# B&R Automation Studio project RobotNewEra (part 4)

```c
	// prepare
	int bol = m_brightleft ? m_elxlist.GetSize() : -1;
	int stp = m_brightleft ? -1 : 1;
	int eol = m_brightleft ? -1 : m_elxlist.GetSize();

	// from last
	int n = eol - stp;

	while(n != bol && ! m_elxlist[n]->MatchNext(pContext))
		n -= stp;

	if(n != bol)
		n += stp;
	else
		return 0;

	// match rest
	while(n != eol)
	{
		if(m_elxlist[n]->Match(pContext))
		{
			n += stp;
		}
		else
		{
			n -= stp;

			while(n != bol && ! m_elxlist[n]->MatchNext(pContext))
				n -= stp;

			if(n != bol)
				n += stp;
			else
				return 0;
		}
	}

	return 1;
}

// mresult.cpp: implementation of the MatchResult class.
//
template <int x> MatchResultT <x> :: MatchResultT(CContext * pContext, int nMaxNumber)
{
	if(pContext != 0)
	{
		m_result.Prepare(nMaxNumber * 2 + 3, -1);

		// matched
		m_result[0] = 1;
		m_result[1] = nMaxNumber;

		for(int n = 0; n <= nMaxNumber; n++)
		{
			int index = pContext->m_captureindex[n];
			//if( index < 0 ) continue;
			if( ! CBracketElxT<char>::CheckCaptureIndex(index, pContext, n) ) continue;

			// check enclosed
			int pos1 = pContext->m_capturestack[index + 1];
			int pos2 = pContext->m_capturestack[index + 2];

			// info
			m_result[n*2 + 2] = pos1 < pos2 ? pos1 : pos2;
			m_result[n*2 + 3] = pos1 < pos2 ? pos2 : pos1;
		}
	}
}

template <int x> inline int MatchResultT <x> :: IsMatched() const
{
	return m_result.At(0, 0);
}

template <int x> inline int MatchResultT <x> :: MaxGroupNumber() const
{
	return m_result.At(1, 0);
}

template <int x> inline int MatchResultT <x> :: GetStart() const
{
	return m_result.At(2, -1);
}

template <int x> inline int MatchResultT <x> :: GetEnd() const
{
	return m_result.At(3, -1);
}

template <int x> inline int MatchResultT <x> :: GetGroupStart(int nGroupNumber) const
{
	return m_result.At(2 + nGroupNumber * 2, -1);
}

template <int x> inline int MatchResultT <x> :: GetGroupEnd(int nGroupNumber) const
{
	return m_result.At(2 + nGroupNumber * 2 + 1, -1);
}

template <int x> MatchResultT <x> & MatchResultT <x> :: operator = (const MatchResultT <x> & result)
{
	m_result.Restore(0);
	if(result.m_result.GetSize() > 0) m_result.Append(result.m_result.GetBuffer(), result.m_result.GetSize());

	return *this;
}

// posselx.cpp: implementation of the CPossessiveElx class.
//
template <int x> CPossessiveElxT <x> :: CPossessiveElxT(ElxInterface * pelx, int nmin, int nmax) : CGreedyElxT <x> (pelx, nmin, nmax)
{
}

template <int x> int CPossessiveElxT <x> :: Match(CContext * pContext) const
{
	int nbegin = pContext->m_nCurrentPos;
	int nsize  = pContext->m_stack.GetSize();
	int ncsize = pContext->m_capturestack.GetSize();
	int bsucc  = 1;

	// match
	if( ! CRepeatElxT <x> :: MatchFixed(pContext) )
	{
		bsucc = 0;
	}
	else
	{
		while( ! CGreedyElxT <x> :: MatchVart(pContext) )
		{
			if( ! CRepeatElxT <x> :: MatchNextFixed(pContext) )
			{
				bsucc = 0;
				break;
			}
		}
	}

	// status
	pContext->m_stack.Restore(nsize);

	if( bsucc )
	{
		pContext->m_stack.Push(nbegin);
		pContext->m_stack.Push(ncsize);
	}

	return bsucc;
}

template <int x> int CPossessiveElxT <x> :: MatchNext(CContext * pContext) const
{
	int nbegin = 0, ncsize = 0;

	pContext->m_stack.Pop(ncsize);
	pContext->m_stack.Pop(nbegin);

	pContext->m_capturestack.Restore(ncsize);
	pContext->m_nCurrentPos = nbegin;

	return 0;
}

// reluctx.cpp: implementation of the CReluctantElx class.
//
template <int x> CReluctantElxT <x> :: CReluctantElxT(ElxInterface * pelx, int nmin, int nmax) : CRepeatElxT <x> (pelx, nmin)
{
	m_nvart = nmax - nmin;
}

template <int x> int CReluctantElxT <x> :: Match(CContext * pContext) const
{
	if( ! CRepeatElxT <x> :: MatchFixed(pContext) )
		return 0;

	while( ! MatchVart(pContext) )
	{
		if( ! CRepeatElxT <x> :: MatchNextFixed(pContext) )
			return 0;
	}

	return 1;
}

template <int x> int CReluctantElxT <x> :: MatchNext(CContext * pContext) const
{
	if( MatchNextVart(pContext) )
		return 1;

	if( ! CRepeatElxT <x> :: MatchNextFixed(pContext) )
		return 0;

	while( ! MatchVart(pContext) )
	{
		if( ! CRepeatElxT <x> :: MatchNextFixed(pContext) )
			return 0;
	}

	return 1;
}

template <int x> int CReluctantElxT <x> :: MatchVart(CContext * pContext) const
{
	pContext->m_stack.Push(0);

	return 1;
}

template <int x> int CReluctantElxT <x> :: MatchNextVart(CContext * pContext) const
{
	int n = 0, nbegin = pContext->m_nCurrentPos;

	pContext->m_stack.Pop(n);

	if(n < m_nvart && CRepeatElxT <x> :: m_pelx->Match(pContext))
	{
		while(pContext->m_nCurrentPos == nbegin)
		{
			if( ! CRepeatElxT <x> :: m_pelx->MatchNext(pContext) ) break;
		}

		if(pContext->m_nCurrentPos != nbegin)
		{
			n ++;

			pContext->m_stack.Push(nbegin);
			pContext->m_stack.Push(n);

			return 1;
		}
	}

	while(n > 0)
	{
		pContext->m_stack.Pop(nbegin);

		while( CRepeatElxT <x> :: m_pelx->MatchNext(pContext) )
		{
			if(pContext->m_nCurrentPos != nbegin)
			{
				pContext->m_stack.Push(nbegin);
				pContext->m_stack.Push(n);

				return 1;
			}
		}

		n --;
	}

	return 0;
}

// repeatx.cpp: implementation of the CRepeatElx class.
//
template <int x> CRepeatElxT <x> :: CRepeatElxT(ElxInterface * pelx, int ntimes)
{
	m_pelx   = pelx;
	m_nfixed = ntimes;
}

template <int x> int CRepeatElxT <x> :: Match(CContext * pContext) const
{
	return MatchFixed(pContext);
}

template <int x> int CRepeatElxT <x> :: MatchNext(CContext * pContext) const
{
	return MatchNextFixed(pContext);
}

template <int x> int CRepeatElxT <x> :: MatchFixed(CContext * pContext) const
{
	if(m_nfixed == 0)
		return 1;

	int n = 0;

	while(n < m_nfixed)
	{
		if(m_pelx->Match(pContext))
		{
			n ++;
		}
		else
		{
			n --;

			while(n >= 0 && ! m_pelx->MatchNext(pContext))
				n --;

			if(n >= 0)
				n ++;
			else
				return 0;
		}
	}

	return 1;
}

template <int x> int CRepeatElxT <x> :: MatchNextFixed(CContext * pContext) const
{
	if(m_nfixed == 0)
		return 0;

	// from last
	int n = m_nfixed - 1;

	while(n >= 0 && ! m_pelx->MatchNext(pContext))
		n --;

	if(n >= 0)
		n ++;
	else
		return 0;

	// match rest
	while(n < m_nfixed)
	{
		if(m_pelx->Match(pContext))
		{
			n ++;
		}
		else
		{
			n --;

			while(n >= 0 && ! m_pelx->MatchNext(pContext))
				n --;

			if(n >= 0)
				n ++;
			else
				return 0;
		}
	}

	return 1;
}

// Regexp
typedef CRegexpT <char> CRegexpA;
typedef CRegexpT <unsigned short> CRegexpW;

#if defined(_UNICODE) || defined(UNICODE)
	typedef CRegexpW CRegexp;
#else
	typedef CRegexpA CRegexp;
#endif

#endif//__DEELX_REGEXP__H__
```

### Package Logical/MotionHandling - Motion Handling

### MotionGlobal.typ
```iecst
(********************************************************************
 * COPYRIGHT -- Bernecker + Rainer
 ********************************************************************
 * File: Global.typ
 * Author: radaka
 * Created: February 09, 2009
 ********************************************************************
 * Global data types of project CncMotionHandling
 ********************************************************************)

TYPE
	ErrorText_Type : 	STRUCT
		Line1 : STRING[79];
		Line2 : STRING[79];
		Line3 : STRING[79];
		Line4 : STRING[79];
	END_STRUCT;
	Error_Type : 	STRUCT
		Count : UINT;
		HmiCount : UINT;
		Class : UINT;
		Number : UDINT;
		Info : ARRAY[0..11]OF USINT;
		Text : ErrorText_Type;
	END_STRUCT;
END_TYPE
```

### MotionGlobalDefines.var
```iecst
(********************************************************************
 * COPYRIGHT -- Bernecker + Rainer
 ********************************************************************
 * File: Global.var
 * Author: radaka
 * Created: February 09, 2009
 ********************************************************************
 * Global variables of project CncMotionHandling
 ********************************************************************)
(*Machine Definitions*)
VAR CONSTANT
	ROBOT : USINT := 0;
END_VAR
(**)
(*Modes Definitions*)
VAR CONSTANT
	MODE_AUTO : USINT := 0;
	MODE_JOG : USINT := 1;
END_VAR
(**)
(*Cnc Definitions*)
VAR CONSTANT
	CNC : USINT := 0;
END_VAR
(**)
(*Axes definitions*)
VAR CONSTANT
	AXIS_X : USINT := 0;
	AXIS_Y : USINT := 1;
	AXIS_Z : USINT := 2;
	AXIS_A : USINT := 3;
	AXIS_B : USINT := 4;
	AXIS_C : USINT := 5;
	AXIS_Q1 : USINT := 6;
	AXIS_Q2 : USINT := 7;
	AXIS_Q3 : USINT := 8;
	AXIS_Q4 : USINT := 9;
	AXIS_Q5 : USINT := 10;
	AXIS_Q6 : USINT := 11;
	AXIS_PS : USINT := 12;
	AXIS_FRAME_X : USINT := 13;
END_VAR
(**)
(*Transformations Definitions*)
VAR
	Robot_TRF : TRF_DATA04_typ;
END_VAR
```

### MotionGlobalSize.var
```iecst
(********************************************************************
 * COPYRIGHT -- Bernecker + Rainer
 ********************************************************************
 * File: Global.var
 * Author: radaka
 * Created: February 09, 2009
 ********************************************************************
 * Global variables of project CncMotionHandling
 ********************************************************************)
VAR CONSTANT
	LABEL_SIZE : USINT := 80;
END_VAR
(********************************************************************
MODE*)
VAR CONSTANT
	MAX_MODE : USINT := 2;
	MAX_MODE_MINUS_ONE : USINT := MAX_MODE-1;
END_VAR
(********************************************************************
SYS*)
VAR CONSTANT
	MAX_SYS : USINT := 1;
	MAX_SYS_MINUS_ONE : USINT := MAX_SYS-1;
END_VAR
(********************************************************************
CNC*)
VAR CONSTANT
	MAX_CNC : USINT := 1;
	MAX_CNC_MINUS_ONE : USINT := MAX_CNC-1;
END_VAR
(********************************************************************
AX*)
VAR CONSTANT
	MAX_AX : USINT := 13; (*6 TCP + 6 JOINTS + 1 PS + 1 FRAME*)
	MAX_AX_MINUS_TWO : USINT := MAX_AX-2;
	MAX_AX_MINUS_ONE : USINT := MAX_AX-1;
END_VAR
```

### Package Logical/MotionHandling/Configuration - GMC

### Config.typ
```iecst
TYPE
	ConfigInputParameter_Type : 	STRUCT
		SimulatedHardwareAR000 : USINT;
		SystemAddress : UDINT;
		CncAddress : UDINT;
		AxesAddress : UDINT;
		TrfAddress : UDINT;
	END_STRUCT;
	ConfigInput_Type : 	STRUCT
		Parameter : ConfigInputParameter_Type;
	END_STRUCT;
	ConfigOutputMonitor_Type : 	STRUCT
		ConfigOk : BOOL;
	END_STRUCT;
	ConfigOutput_Type : 	STRUCT
		Monitor : ConfigOutputMonitor_Type;
	END_STRUCT;
	Config_Type : 	STRUCT
		Input : ConfigInput_Type;
		Output : ConfigOutput_Type;
	END_STRUCT;
END_TYPE
```

### Program Logical/MotionHandling/Configuration/Config (IEC) - Configuration Of GMC

#### ConfigActions.st
```iecst
(********************************************************************
 * COPYRIGHT -- Bernecker + Rainer
 ********************************************************************
 * Program: Config
 * File: DefaultConfig.st
 * Author: radaka
 * Created: February 18, 2009
 ********************************************************************
 * Implementation of program Config
 ********************************************************************)

ACTION Configuration_Prepare:

	(* Loop over all systems *)
	FOR i:= 0 TO MAX_SYS_MINUS_ONE DO

		FOR j:= 0 TO MAX_AX_MINUS_ONE DO
			pSystem[i].Input.Configuration.SystemAxes[j].Index:= NO_PART_OF_SYSTEM;
			pSystem[i].Input.Configuration.SystemPowerAxesIndex[j]:= NO_PART_OF_SYSTEM;
		END_FOR
		FOR j:= 0 TO MAX_CNC_MINUS_ONE DO
			pSystem[i].Input.Configuration.SystemCncIndex[j]:= NO_PART_OF_SYSTEM;
		END_FOR

		FOR j:= 0 TO MAX_MODE_MINUS_ONE DO
			FOR k:= 0 TO MAX_CNC_MINUS_ONE DO
				pSystem[i].Input.Configuration.Mode[j].Cnc[k].Index:= NO_PART_OF_SYSTEM;
			END_FOR
			FOR k:= 0 TO MAX_AX_MINUS_ONE DO
				pSystem[i].Input.Configuration.Mode[j].Axes[k].Index:= NO_PART_OF_SYSTEM;
			END_FOR
		END_FOR

	(* End Loop over all systems *)
	END_FOR

END_ACTION

ACTION CNCConfig:

		(********************************************************************************************************)
		(* System Configuration *)

	pSystem[ROBOT].Input.Configuration.Active := 1;
	pSystem[ROBOT].Input.Configuration.Label := 'Robot';

	pSystem[ROBOT].Input.Configuration.SystemCncIndex[0] := CNC;

	pSystem[ROBOT].Input.Configuration.SystemPowerAxesIndex[0] := AXIS_PS;

	pSystem[ROBOT].Input.Configuration.SystemAxes[0].Index:= AXIS_X;
	pSystem[ROBOT].Input.Configuration.SystemAxes[0].HomeOrder:= 1;
	pSystem[ROBOT].Input.Configuration.SystemAxes[1].Index:= AXIS_Y;
	pSystem[ROBOT].Input.Configuration.SystemAxes[1].HomeOrder:= 1;
	pSystem[ROBOT].Input.Configuration.SystemAxes[2].Index:= AXIS_Z;
	pSystem[ROBOT].Input.Configuration.SystemAxes[2].HomeOrder:= 1;
	pSystem[ROBOT].Input.Configuration.SystemAxes[3].Index:= AXIS_A;
	pSystem[ROBOT].Input.Configuration.SystemAxes[3].HomeOrder:= 1;
	pSystem[ROBOT].Input.Configuration.SystemAxes[4].Index:= AXIS_B;
	pSystem[ROBOT].Input.Configuration.SystemAxes[4].HomeOrder:= 1;
	pSystem[ROBOT].Input.Configuration.SystemAxes[5].Index:= AXIS_C;
	pSystem[ROBOT].Input.Configuration.SystemAxes[5].HomeOrder:= 1;

	pSystem[ROBOT].Input.Configuration.SystemAxes[6].Index:= AXIS_Q1;
	pSystem[ROBOT].Input.Configuration.SystemAxes[6].HomeOrder:= 0;
	pSystem[ROBOT].Input.Configuration.SystemAxes[7].Index:= AXIS_Q2;
	pSystem[ROBOT].Input.Configuration.SystemAxes[7].HomeOrder:= 0;
	pSystem[ROBOT].Input.Configuration.SystemAxes[8].Index:= AXIS_Q3;
	pSystem[ROBOT].Input.Configuration.SystemAxes[8].HomeOrder:= 0;
	pSystem[ROBOT].Input.Configuration.SystemAxes[9].Index:= AXIS_Q4;
	pSystem[ROBOT].Input.Configuration.SystemAxes[9].HomeOrder:= 0;
	pSystem[ROBOT].Input.Configuration.SystemAxes[10].Index:= AXIS_Q5;
	pSystem[ROBOT].Input.Configuration.SystemAxes[10].HomeOrder:= 0;
	pSystem[ROBOT].Input.Configuration.SystemAxes[11].Index:= AXIS_Q6;
	pSystem[ROBOT].Input.Configuration.SystemAxes[11].HomeOrder:= 0;

	(********************************************************************************************************)
	(* Mode Configuration - CNC  *)
	pSystem[ROBOT].Input.Configuration.Mode[MODE_AUTO].Cnc[0].Index:= CNC;
	pSystem[ROBOT].Input.Configuration.Mode[MODE_AUTO].Cnc[0].Behavior:= STOP_CNC;
	pSystem[ROBOT].Input.Configuration.Mode[MODE_AUTO].Cnc[0].Visible:= 1;

	pSystem[ROBOT].Input.Configuration.Mode[MODE_AUTO].Axes[0].Index:= AXIS_X;
	pSystem[ROBOT].Input.Configuration.Mode[MODE_AUTO].Axes[0].Type:= CNC_AXES;
	pSystem[ROBOT].Input.Configuration.Mode[MODE_AUTO].Axes[0].Behavior:= HOMEAUTO_AXES;
	pSystem[ROBOT].Input.Configuration.Mode[MODE_AUTO].Axes[0].Visible:= 1;

	pSystem[ROBOT].Input.Configuration.Mode[MODE_AUTO].Axes[1].Index:= AXIS_Y;
	pSystem[ROBOT].Input.Configuration.Mode[MODE_AUTO].Axes[1].Type:= CNC_AXES;
	pSystem[ROBOT].Input.Configuration.Mode[MODE_AUTO].Axes[1].Behavior:= HOMEAUTO_AXES;
	pSystem[ROBOT].Input.Configuration.Mode[MODE_AUTO].Axes[1].Visible:= 1;

	pSystem[ROBOT].Input.Configuration.Mode[MODE_AUTO].Axes[2].Index:= AXIS_Z;
	pSystem[ROBOT].Input.Configuration.Mode[MODE_AUTO].Axes[2].Type:= CNC_AXES;
	pSystem[ROBOT].Input.Configuration.Mode[MODE_AUTO].Axes[2].Behavior:= HOMEAUTO_AXES;
	pSystem[ROBOT].Input.Configuration.Mode[MODE_AUTO].Axes[2].Visible:= 1;

	pSystem[ROBOT].Input.Configuration.Mode[MODE_AUTO].Axes[3].Index:= AXIS_A;
	pSystem[ROBOT].Input.Configuration.Mode[MODE_AUTO].Axes[3].Type:= CNC_AXES;
	pSystem[ROBOT].Input.Configuration.Mode[MODE_AUTO].Axes[3].Behavior:= HOMEAUTO_AXES;
	pSystem[ROBOT].Input.Configuration.Mode[MODE_AUTO].Axes[3].Visible:= 1;

	pSystem[ROBOT].Input.Configuration.Mode[MODE_AUTO].Axes[4].Index:= AXIS_B;
	pSystem[ROBOT].Input.Configuration.Mode[MODE_AUTO].Axes[4].Type:= CNC_AXES;
	pSystem[ROBOT].Input.Configuration.Mode[MODE_AUTO].Axes[4].Behavior:= HOMEAUTO_AXES;
	pSystem[ROBOT].Input.Configuration.Mode[MODE_AUTO].Axes[4].Visible:= 1;

	pSystem[ROBOT].Input.Configuration.Mode[MODE_AUTO].Axes[5].Index:= AXIS_C;
	pSystem[ROBOT].Input.Configuration.Mode[MODE_AUTO].Axes[5].Type:= CNC_AXES;
	pSystem[ROBOT].Input.Configuration.Mode[MODE_AUTO].Axes[5].Behavior:= HOMEAUTO_AXES;
	pSystem[ROBOT].Input.Configuration.Mode[MODE_AUTO].Axes[5].Visible:= 1;

	pSystem[ROBOT].Input.Configuration.Mode[MODE_AUTO].Axes[6].Index:= AXIS_Q1;
	pSystem[ROBOT].Input.Configuration.Mode[MODE_AUTO].Axes[6].Type:= CNC_AXES;
	pSystem[ROBOT].Input.Configuration.Mode[MODE_AUTO].Axes[6].Behavior:= STOP_AXES;
	pSystem[ROBOT].Input.Configuration.Mode[MODE_AUTO].Axes[6].Visible:= 1;

	pSystem[ROBOT].Input.Configuration.Mode[MODE_AUTO].Axes[7].Index:= AXIS_Q2;
	pSystem[ROBOT].Input.Configuration.Mode[MODE_AUTO].Axes[7].Type:= CNC_AXES;
	pSystem[ROBOT].Input.Configuration.Mode[MODE_AUTO].Axes[7].Behavior:= STOP_AXES;
	pSystem[ROBOT].Input.Configuration.Mode[MODE_AUTO].Axes[7].Visible:= 1;

	pSystem[ROBOT].Input.Configuration.Mode[MODE_AUTO].Axes[8].Index:= AXIS_Q3;
	pSystem[ROBOT].Input.Configuration.Mode[MODE_AUTO].Axes[8].Type:= CNC_AXES;
	pSystem[ROBOT].Input.Configuration.Mode[MODE_AUTO].Axes[8].Behavior:= STOP_AXES;
	pSystem[ROBOT].Input.Configuration.Mode[MODE_AUTO].Axes[8].Visible:= 1;

	pSystem[ROBOT].Input.Configuration.Mode[MODE_AUTO].Axes[9].Index:= AXIS_Q4;
	pSystem[ROBOT].Input.Configuration.Mode[MODE_AUTO].Axes[9].Type:= CNC_AXES;
	pSystem[ROBOT].Input.Configuration.Mode[MODE_AUTO].Axes[9].Behavior:= STOP_AXES;
	pSystem[ROBOT].Input.Configuration.Mode[MODE_AUTO].Axes[9].Visible:= 1;

	pSystem[ROBOT].Input.Configuration.Mode[MODE_AUTO].Axes[10].Index:= AXIS_Q5;
	pSystem[ROBOT].Input.Configuration.Mode[MODE_AUTO].Axes[10].Type:= CNC_AXES;
	pSystem[ROBOT].Input.Configuration.Mode[MODE_AUTO].Axes[10].Behavior:= STOP_AXES;
	pSystem[ROBOT].Input.Configuration.Mode[MODE_AUTO].Axes[10].Visible:= 1;

	pSystem[ROBOT].Input.Configuration.Mode[MODE_AUTO].Axes[11].Index:= AXIS_Q6;
	pSystem[ROBOT].Input.Configuration.Mode[MODE_AUTO].Axes[11].Type:= CNC_AXES;
	pSystem[ROBOT].Input.Configuration.Mode[MODE_AUTO].Axes[11].Behavior:= STOP_AXES;
	pSystem[ROBOT].Input.Configuration.Mode[MODE_AUTO].Axes[11].Visible:= 1;

	(********************************************************************************************************)
	(* Mode Configuration - AXES  *)
	pSystem[ROBOT].Input.Configuration.Mode[MODE_JOG].Cnc[0].Index:= CNC;
	pSystem[ROBOT].Input.Configuration.Mode[MODE_JOG].Cnc[0].Behavior:= STOP_CNC;
	pSystem[ROBOT].Input.Configuration.Mode[MODE_JOG].Cnc[0].Visible:= 0;

	pSystem[ROBOT].Input.Configuration.Mode[MODE_JOG].Axes[0].Index:= AXIS_X;
	pSystem[ROBOT].Input.Configuration.Mode[MODE_JOG].Axes[0].Type:= AUXILIARY_AXES;
	pSystem[ROBOT].Input.Configuration.Mode[MODE_JOG].Axes[0].Behavior:= STOP_AXES;
	pSystem[ROBOT].Input.Configuration.Mode[MODE_JOG].Axes[0].Visible:= 0;

	pSystem[ROBOT].Input.Configuration.Mode[MODE_JOG].Axes[1].Index:= AXIS_Y;
	pSystem[ROBOT].Input.Configuration.Mode[MODE_JOG].Axes[1].Type:= AUXILIARY_AXES;
	pSystem[ROBOT].Input.Configuration.Mode[MODE_JOG].Axes[1].Behavior:= STOP_AXES;
	pSystem[ROBOT].Input.Configuration.Mode[MODE_JOG].Axes[1].Visible:= 0;

	pSystem[ROBOT].Input.Configuration.Mode[MODE_JOG].Axes[2].Index:= AXIS_Z;
	pSystem[ROBOT].Input.Configuration.Mode[MODE_JOG].Axes[2].Type:= AUXILIARY_AXES;
	pSystem[ROBOT].Input.Configuration.Mode[MODE_JOG].Axes[2].Behavior:= STOP_AXES;
	pSystem[ROBOT].Input.Configuration.Mode[MODE_JOG].Axes[2].Visible:= 0;

	pSystem[ROBOT].Input.Configuration.Mode[MODE_JOG].Axes[3].Index:= AXIS_A;
	pSystem[ROBOT].Input.Configuration.Mode[MODE_JOG].Axes[3].Type:= AUXILIARY_AXES;
	pSystem[ROBOT].Input.Configuration.Mode[MODE_JOG].Axes[3].Behavior:= STOP_AXES;
	pSystem[ROBOT].Input.Configuration.Mode[MODE_JOG].Axes[3].Visible:= 0;

	pSystem[ROBOT].Input.Configuration.Mode[MODE_JOG].Axes[4].Index:= AXIS_B;
	pSystem[ROBOT].Input.Configuration.Mode[MODE_JOG].Axes[4].Type:= AUXILIARY_AXES;
	pSystem[ROBOT].Input.Configuration.Mode[MODE_JOG].Axes[4].Behavior:= STOP_AXES;
	pSystem[ROBOT].Input.Configuration.Mode[MODE_JOG].Axes[4].Visible:= 0;

	pSystem[ROBOT].Input.Configuration.Mode[MODE_JOG].Axes[5].Index:= AXIS_C;
	pSystem[ROBOT].Input.Configuration.Mode[MODE_JOG].Axes[5].Type:= AUXILIARY_AXES;
	pSystem[ROBOT].Input.Configuration.Mode[MODE_JOG].Axes[5].Behavior:= STOP_AXES;
	pSystem[ROBOT].Input.Configuration.Mode[MODE_JOG].Axes[5].Visible:= 0;

	pSystem[ROBOT].Input.Configuration.Mode[MODE_JOG].Axes[6].Index:= AXIS_Q1;
	pSystem[ROBOT].Input.Configuration.Mode[MODE_JOG].Axes[6].Type:= JOG_AXES;
	pSystem[ROBOT].Input.Configuration.Mode[MODE_JOG].Axes[6].Behavior:= STOP_AXES;
	pSystem[ROBOT].Input.Configuration.Mode[MODE_JOG].Axes[6].Visible:= 1;

	pSystem[ROBOT].Input.Configuration.Mode[MODE_JOG].Axes[7].Index:= AXIS_Q2;
	pSystem[ROBOT].Input.Configuration.Mode[MODE_JOG].Axes[7].Type:= JOG_AXES;
	pSystem[ROBOT].Input.Configuration.Mode[MODE_JOG].Axes[7].Behavior:= STOP_AXES;
	pSystem[ROBOT].Input.Configuration.Mode[MODE_JOG].Axes[7].Visible:= 1;

	pSystem[ROBOT].Input.Configuration.Mode[MODE_JOG].Axes[8].Index:= AXIS_Q3;
	pSystem[ROBOT].Input.Configuration.Mode[MODE_JOG].Axes[8].Type:= JOG_AXES;
	pSystem[ROBOT].Input.Configuration.Mode[MODE_JOG].Axes[8].Behavior:= STOP_AXES;
	pSystem[ROBOT].Input.Configuration.Mode[MODE_JOG].Axes[8].Visible:= 1;

	pSystem[ROBOT].Input.Configuration.Mode[MODE_JOG].Axes[9].Index:= AXIS_Q4;
	pSystem[ROBOT].Input.Configuration.Mode[MODE_JOG].Axes[9].Type:= JOG_AXES;
	pSystem[ROBOT].Input.Configuration.Mode[MODE_JOG].Axes[9].Behavior:= STOP_AXES;
	pSystem[ROBOT].Input.Configuration.Mode[MODE_JOG].Axes[9].Visible:= 1;

	pSystem[ROBOT].Input.Configuration.Mode[MODE_JOG].Axes[10].Index:= AXIS_Q5;
	pSystem[ROBOT].Input.Configuration.Mode[MODE_JOG].Axes[10].Type:= JOG_AXES;
	pSystem[ROBOT].Input.Configuration.Mode[MODE_JOG].Axes[10].Behavior:= STOP_AXES;
	pSystem[ROBOT].Input.Configuration.Mode[MODE_JOG].Axes[10].Visible:= 1;

	pSystem[ROBOT].Input.Configuration.Mode[MODE_JOG].Axes[11].Index:= AXIS_Q6;
	pSystem[ROBOT].Input.Configuration.Mode[MODE_JOG].Axes[11].Type:= JOG_AXES;
	pSystem[ROBOT].Input.Configuration.Mode[MODE_JOG].Axes[11].Behavior:= STOP_AXES;
	pSystem[ROBOT].Input.Configuration.Mode[MODE_JOG].Axes[11].Visible:= 1;

	//		(********************************************************************************************************)
	(* Cnc Configuration *)
	pCnc[CNC].Input.Configuration.Active:= 1;
	pCnc[CNC].Input.Configuration.NcMapObjName:= 'gRobot';
	pCnc[CNC].Input.Configuration.Warnings:= ncOFF;
	pCnc[CNC].Input.Configuration.ErrorTextDataModulName:= 'arnc0001';

	(********************************************************************************************************)
	(* Axes Configuration *)

	pAxes[AXIS_X].Input.Configuration.Active:= 1;
	pAxes[AXIS_X].Input.Configuration.NcMapObjName:= 'gAxisX';
	pAxes[AXIS_X].Input.Configuration.ErrorDatObjName:= 'AcpError';
	pAxes[AXIS_X].Input.Configuration.Label			 := 'X';
	pAxes[AXIS_X].Input.Configuration.UnitPositionFaktor:= 1000;
	pAxes[AXIS_X].Input.Configuration.UnitVelocityFaktor:= 1000;
	pAxes[AXIS_X].Input.Configuration.UnitPositionLabel	:= 'mm';

	pAxes[AXIS_Y].Input.Configuration.Active:= 1;
	pAxes[AXIS_Y].Input.Configuration.NcMapObjName:= 'gAxisY';
	pAxes[AXIS_Y].Input.Configuration.ErrorDatObjName:= 'AcpError';
	pAxes[AXIS_Y].Input.Configuration.Label			 := 'Y';
	pAxes[AXIS_Y].Input.Configuration.UnitPositionFaktor:= 1000;
	pAxes[AXIS_Y].Input.Configuration.UnitVelocityFaktor:= 1000;
	pAxes[AXIS_Y].Input.Configuration.UnitPositionLabel	:= 'mm';

	pAxes[AXIS_Z].Input.Configuration.Active:= 1;
	pAxes[AXIS_Z].Input.Configuration.NcMapObjName:= 'gAxisZ';
	pAxes[AXIS_Z].Input.Configuration.ErrorDatObjName:= 'AcpError';
	pAxes[AXIS_Z].Input.Configuration.Label			 := 'Z';
	pAxes[AXIS_Z].Input.Configuration.UnitPositionFaktor:= 1000;
	pAxes[AXIS_Z].Input.Configuration.UnitVelocityFaktor:= 1000;
	pAxes[AXIS_Z].Input.Configuration.UnitPositionLabel	:= 'mm';

	pAxes[AXIS_A].Input.Configuration.Active:= 1;
	pAxes[AXIS_A].Input.Configuration.NcMapObjName:= 'gAxisA';
	pAxes[AXIS_A].Input.Configuration.ErrorDatObjName:= 'AcpError';
	pAxes[AXIS_A].Input.Configuration.Label			 := 'A';
	pAxes[AXIS_A].Input.Configuration.UnitPositionFaktor:= 1000;
	pAxes[AXIS_A].Input.Configuration.UnitVelocityFaktor:= 1000;
	pAxes[AXIS_A].Input.Configuration.UnitPositionLabel	:= 'mm';

	pAxes[AXIS_B].Input.Configuration.Active:= 1;
	pAxes[AXIS_B].Input.Configuration.NcMapObjName:= 'gAxisB';
	pAxes[AXIS_B].Input.Configuration.ErrorDatObjName:= 'AcpError';
	pAxes[AXIS_B].Input.Configuration.Label			 := 'B';
	pAxes[AXIS_B].Input.Configuration.UnitPositionFaktor:= 1000;
	pAxes[AXIS_B].Input.Configuration.UnitVelocityFaktor:= 1000;
	pAxes[AXIS_B].Input.Configuration.UnitPositionLabel	:= 'mm';

	pAxes[AXIS_C].Input.Configuration.Active:= 1;
	pAxes[AXIS_C].Input.Configuration.NcMapObjName:= 'gAxisC';
	pAxes[AXIS_C].Input.Configuration.ErrorDatObjName:= 'AcpError';
	pAxes[AXIS_C].Input.Configuration.Label			 := 'C';
	pAxes[AXIS_C].Input.Configuration.UnitPositionFaktor:= 1000;
	pAxes[AXIS_C].Input.Configuration.UnitVelocityFaktor:= 1000;
	pAxes[AXIS_C].Input.Configuration.UnitPositionLabel	:= 'mm';

	pAxes[AXIS_Q1].Input.Configuration.Active:= 1;
	pAxes[AXIS_Q1].Input.Configuration.NcMapObjName:= 'gAxisQ1';
	pAxes[AXIS_Q1].Input.Configuration.ErrorDatObjName:= 'AcpError';
	pAxes[AXIS_Q1].Input.Configuration.Label			 := 'J1';
	pAxes[AXIS_Q1].Input.Configuration.UnitPositionFaktor:= 1000;
	pAxes[AXIS_Q1].Input.Configuration.UnitVelocityFaktor:= 1000;
	pAxes[AXIS_Q1].Input.Configuration.UnitPositionLabel	:= 'deg';
//	(* Uncomment the 2 lines under for real machine *)
//	pAxes[AXIS_Q1].Input.Configuration.PDOWriteParID[0] := 247;
//	pAxes[AXIS_Q1].Input.Configuration.PDOWriteParType[0] := 8;
//	pAxes[AXIS_Q1].Input.Configuration.PDOReadParID[0] := 111;
//	pAxes[AXIS_Q1].Input.Configuration.PDOReadParType[0] := ncPAR_TYP_DINT;
//	pAxes[AXIS_Q1].Input.Configuration.PDOReadParID[1] := 113;
//	pAxes[AXIS_Q1].Input.Configuration.PDOReadParType[1] := ncPAR_TYP_DINT;
//	pAxes[AXIS_Q1].Input.Configuration.PDOReadParID[2] := 277;
//	pAxes[AXIS_Q1].Input.Configuration.PDOReadParType[2] := ncPAR_TYP_REAL;

	pAxes[AXIS_Q2].Input.Configuration.Active:= 1;
	pAxes[AXIS_Q2].Input.Configuration.NcMapObjName:= 'gAxisQ2';
	pAxes[AXIS_Q2].Input.Configuration.ErrorDatObjName:= 'AcpError';
	pAxes[AXIS_Q2].Input.Configuration.Label			 := 'J2';
	pAxes[AXIS_Q2].Input.Configuration.UnitPositionFaktor:= 1000;
	pAxes[AXIS_Q2].Input.Configuration.UnitVelocityFaktor:= 1000;
	pAxes[AXIS_Q2].Input.Configuration.UnitPositionLabel	:= 'deg';
(* Uncomment the 2 lines under for real machine *)
//	pAxes[AXIS_Q2].Input.Configuration.PDOWriteParID[0] := 247;
//	pAxes[AXIS_Q2].Input.Configuration.PDOWriteParType[0] := 8;
//	pAxes[AXIS_Q2].Input.Configuration.PDOReadParID[0] := 111;
//	pAxes[AXIS_Q2].Input.Configuration.PDOReadParType[0] := ncPAR_TYP_DINT;
//	pAxes[AXIS_Q2].Input.Configuration.PDOReadParID[1] := 113;
//	pAxes[AXIS_Q2].Input.Configuration.PDOReadParType[1] := ncPAR_TYP_DINT;
//	pAxes[AXIS_Q2].Input.Configuration.PDOReadParID[2] := 277;
//	pAxes[AXIS_Q2].Input.Configuration.PDOReadParType[2] := ncPAR_TYP_REAL;

	pAxes[AXIS_Q3].Input.Configuration.Active:= 1;
	pAxes[AXIS_Q3].Input.Configuration.NcMapObjName:= 'gAxisQ3';
	pAxes[AXIS_Q3].Input.Configuration.ErrorDatObjName:= 'AcpError';
	pAxes[AXIS_Q3].Input.Configuration.Label			 := 'J3';
	pAxes[AXIS_Q3].Input.Configuration.UnitPositionFaktor:= 1000;
	pAxes[AXIS_Q3].Input.Configuration.UnitVelocityFaktor:= 1000;
	pAxes[AXIS_Q3].Input.Configuration.UnitPositionLabel	:= 'deg';
	(* Uncomment the 2 lines under for real machine *)
//	pAxes[AXIS_Q3].Input.Configuration.PDOWriteParID[0] := 247;
//	pAxes[AXIS_Q3].Input.Configuration.PDOWriteParType[0] := 8;
//		pAxes[AXIS_Q3].Input.Configuration.PDOReadParID[0] := 111;
//		pAxes[AXIS_Q3].Input.Configuration.PDOReadParType[0] := ncPAR_TYP_DINT;
//		pAxes[AXIS_Q3].Input.Configuration.PDOReadParID[1] := 113;
//		pAxes[AXIS_Q3].Input.Configuration.PDOReadParType[1] := ncPAR_TYP_DINT;
//		pAxes[AXIS_Q3].Input.Configuration.PDOReadParID[2] := 277;
//		pAxes[AXIS_Q3].Input.Configuration.PDOReadParType[2] := ncPAR_TYP_REAL;

	pAxes[AXIS_Q4].Input.Configuration.Active:= 1;
	pAxes[AXIS_Q4].Input.Configuration.NcMapObjName:= 'gAxisQ4';
	pAxes[AXIS_Q4].Input.Configuration.ErrorDatObjName:= 'AcpError';
	pAxes[AXIS_Q4].Input.Configuration.Label			 := 'J4';
	pAxes[AXIS_Q4].Input.Configuration.UnitPositionFaktor:= 1000;
	pAxes[AXIS_Q4].Input.Configuration.UnitVelocityFaktor:= 1000;
	pAxes[AXIS_Q4].Input.Configuration.UnitPositionLabel	:= 'deg';
//	(* Uncomment the 2 lines under for real machine *)
//	pAxes[AXIS_Q4].Input.Configuration.PDOWriteParID[0] := 247;
//	pAxes[AXIS_Q4].Input.Configuration.PDOWriteParType[0] := 8;
//		pAxes[AXIS_Q4].Input.Configuration.PDOReadParID[0] := 111;
//		pAxes[AXIS_Q4].Input.Configuration.PDOReadParType[0] := ncPAR_TYP_DINT;
//		pAxes[AXIS_Q4].Input.Configuration.PDOReadParID[1] := 113;
//		pAxes[AXIS_Q4].Input.Configuration.PDOReadParType[1] := ncPAR_TYP_DINT;
//		pAxes[AXIS_Q4].Input.Configuration.PDOReadParID[2] := 277;
//		pAxes[AXIS_Q4].Input.Configuration.PDOReadParType[2] := ncPAR_TYP_REAL;

	pAxes[AXIS_Q5].Input.Configuration.Active:= 1;
	pAxes[AXIS_Q5].Input.Configuration.NcMapObjName:= 'gAxisQ5';
	pAxes[AXIS_Q5].Input.Configuration.ErrorDatObjName:= 'AcpError';
	pAxes[AXIS_Q5].Input.Configuration.Label			 := 'J5';
	pAxes[AXIS_Q5].Input.Configuration.UnitPositionFaktor:= 1000;
	pAxes[AXIS_Q5].Input.Configuration.UnitVelocityFaktor:= 1000;
	pAxes[AXIS_Q5].Input.Configuration.UnitPositionLabel	:= 'deg';
	(* Uncomment the 2 lines under for real machine *)
//	pAxes[AXIS_Q5].Input.Configuration.PDOWriteParID[0] := 247;
//	pAxes[AXIS_Q5].Input.Configuration.PDOWriteParType[0] := 8;
//		pAxes[AXIS_Q5].Input.Configuration.PDOReadParID[0] := 111;
//		pAxes[AXIS_Q5].Input.Configuration.PDOReadParType[0] := ncPAR_TYP_DINT;
//		pAxes[AXIS_Q5].Input.Configuration.PDOReadParID[1] := 113;
//		pAxes[AXIS_Q5].Input.Configuration.PDOReadParType[1] := ncPAR_TYP_DINT;
//		pAxes[AXIS_Q5].Input.Configuration.PDOReadParID[2] := 277;
//		pAxes[AXIS_Q5].Input.Configuration.PDOReadParType[2] := ncPAR_TYP_REAL;

	pAxes[AXIS_Q6].Input.Configuration.Active:= 1;
	pAxes[AXIS_Q6].Input.Configuration.NcMapObjName:= 'gAxisQ6';
	pAxes[AXIS_Q6].Input.Configuration.ErrorDatObjName:= 'AcpError';
	pAxes[AXIS_Q6].Input.Configuration.Label			 := 'J6';
	pAxes[AXIS_Q6].Input.Configuration.UnitPositionFaktor:= 1000;
	pAxes[AXIS_Q6].Input.Configuration.UnitVelocityFaktor:= 1000;
	pAxes[AXIS_Q6].Input.Configuration.UnitPositionLabel	:= 'deg';
//	(* Uncomment the 2 lines under for real machine *)
//	pAxes[AXIS_Q6].Input.Configuration.PDOWriteParID[0] := 247;
//	pAxes[AXIS_Q6].Input.Configuration.PDOWriteParType[0] := 8;
//		pAxes[AXIS_Q6].Input.Configuration.PDOReadParID[0] := 111;
//		pAxes[AXIS_Q6].Input.Configuration.PDOReadParType[0] := ncPAR_TYP_DINT;
//		pAxes[AXIS_Q6].Input.Configuration.PDOReadParID[1] := 113;
//		pAxes[AXIS_Q6].Input.Configuration.PDOReadParType[1] := ncPAR_TYP_DINT;
//		pAxes[AXIS_Q6].Input.Configuration.PDOReadParID[2] := 277;
//		pAxes[AXIS_Q6].Input.Configuration.PDOReadParType[2] := ncPAR_TYP_REAL;

	pAxes[AXIS_PS].Input.Configuration.Active:= 1;
	pAxes[AXIS_PS].Input.Configuration.NcMapObjName:= 'gPowerSupply';
	pAxes[AXIS_PS].Input.Configuration.ErrorDatObjName:= 'AcpError';
	pAxes[AXIS_PS].Input.Configuration.Label			 := 'AXIS_PS';
	pAxes[AXIS_PS].Input.Configuration.UnitPositionFaktor:= 1000;
	pAxes[AXIS_PS].Input.Configuration.UnitVelocityFaktor:= 1000;

	//pAxes[AXIS_FRAME_X].Input.Configuration.Active:= 1;
	//pAxes[AXIS_FRAME_X].Input.Configuration.NcMapObjName:= 'gAxisFrameX';
	//pAxes[AXIS_FRAME_X].Input.Configuration.ErrorDatObjName:= 'AcpError';
	//pAxes[AXIS_FRAME_X].Input.Configuration.UnitPositionFaktor:= 1000;
	//pAxes[AXIS_FRAME_X].Input.Configuration.UnitVelocityFaktor:= 1000;

	(********************************************************************************************************)

END_ACTION

ACTION InitAxesObj:
	gAxisQ1;
	gAxisQ2;
	gAxisQ3;
	gAxisQ4;
	gAxisQ5;
	gAxisQ6;
	gAxisX;
	gAxisY;
	gAxisZ;
	gAxisA;
	gAxisB;
	gAxisC;
END_ACTION

ACTION InitCncObj:

	gRobot;

END_ACTION
```

#### Config.st - Initialization code
```iecst
(********************************************************************
 * COPYRIGHT -- Bernecker + Rainer
 ********************************************************************
 * Program: Configuration
 * File: Config.st
 * Author: radaka
 * Created: February 18, 2009
 ********************************************************************
 * Implementation of program Configuration
 ********************************************************************)

PROGRAM _INIT

	Config.Output.Monitor.ConfigOk:= 0;
	InitAxesObj;
	InitCncObj;
END_PROGRAM

PROGRAM _CYCLIC

	Config.Input.Parameter.AxesAddress := HmiGlobal.Address.AxesAddress;
	Config.Input.Parameter.CncAddress := HmiGlobal.Address.CncAddress;
	Config.Input.Parameter.SystemAddress := HmiGlobal.Address.SystemAddress;

	IF	(Config.Input.Parameter.AxesAddress <> 0) AND
 		(Config.Input.Parameter.CncAddress <> 0)AND
  		(Config.Input.Parameter.SystemAddress <> 0) THEN

		pAxes ACCESS Config.Input.Parameter.AxesAddress;
		pCnc ACCESS Config.Input.Parameter.CncAddress;
  		pSystem ACCESS Config.Input.Parameter.SystemAddress;

  		IF(Config.Output.Monitor.ConfigOk = 0)THEN

			(********************************************************************************************************)
			(* Preparation of the configuration *)
			Configuration_Prepare;
			(********************************************************************************************************)

			CNCConfig;

			(********************************************************************************************************)
			Config.Output.Monitor.ConfigOk:= TRUE;
			(********************************************************************************************************)
		END_IF

	END_IF

END_PROGRAM
```

#### Config.var
```iecst
(********************************************************************
 * COPYRIGHT -- Bernecker + Rainer
 ********************************************************************
 * Program: Axes
 * File: Axes.var
 * Author: radaka
 * Created: February 09, 2009
 ********************************************************************
 * Local variables of program Axes
 ********************************************************************)
VAR
	i : USINT;
	j : USINT;
	k : USINT;
	Config : Config_Type := (0);
	pAxes : REFERENCE TO ARRAY[0..MAX_AX_MINUS_ONE] OF Axes_Type;
	pCnc : REFERENCE TO ARRAY[0..MAX_CNC_MINUS_ONE] OF Cnc_Type;
	pSystem : REFERENCE TO ARRAY[0..MAX_SYS_MINUS_ONE] OF System_Type;
END_VAR
```

### Package Logical/MotionHandling/SystemHandling - GMC

### System.typ - Local data types
```iecst
(********************************************************************
 * COPYRIGHT -- Bernecker + Rainer
 ********************************************************************
 * Program: System
 * File: System.typ
 * Author: radaka
 * Created: February 18, 2009
 ********************************************************************
 * Local data types of program System
 ********************************************************************)

TYPE
	System_Type : 	STRUCT
		Input : SystemInput_Type; (*Input structure*)
		Output : SystemOutput_Type; (*Output structure*)
	END_STRUCT;
	SystemInConfModeAxBehav_Type :
		(
		STOP_AXES, (*Axis with this behavior will be stopped during modechange.*)
		IGNORE_AXES, (*Axes with this behavior will be ingnored during Modechange. This is the only behavior without stopping the axis*)
		HOMEAUTO_AXES, (*Axes with this behavior will be direct homed to their AutoPosition parameter during Modechange*)
		HOMEAUTO_MOVE_AXES, (*Axes with this behavior will be direct homed to their AutoPosition Paramter and then ablsolute moved to the Position parameter during Modechange*)
		HOMEAUTO_CYCLICPOS_AXES, (*Axes with this behavior will be direct homed to their AutoPosition Paramter and then linked to their CyclicPosition parameter during Modechange*)
		HOMEAUTO_MOVE_CYCLICPOS_AXES, (*Axes with this behavior will be direct homed to their AutoPosition Paramter, absolute moved to the Position parameter and then linked to their CyclicPosition parameter during Modechange*)
		MOVE_AXES, (*Axes with this behavior will be absolute moved to their Position parameter during Modechange*)
		MOVE_HOMEAUTO_AXES, (*Axes with this behavior will be absolute moved to their Position parameter and then direct homed to their AutoPosition parameter during Modechange*)
		MOVE_HOMEAUTO_CYCLICPOS_AXES, (*Axes with this behavior will be absolute moved to their Position parameter, direct homed to their AutoPosition parameter and then linked to their CyclicPosition parameter during Modechange*)
		MOVE_CYCLICPOS_AXES, (*Axes with this behavior will be absolute moved to their Position parameter and then linked to their CyclicPosition parameter during Modechange*)
		CYCLICPOS_AXES (*Axes with this behavior will be linked to their CyclicPosition parameter during Modechange*)
		);
	SystemInConfModeCncBehav_Type :
		(
		STOP_CNC,
		IGNORE_CNC
		);
	SystemInput_Type : 	STRUCT
		Configuration : SystemInputConfiguration_Type; (*Configuration*)
		Command : SystemInputCommand_Type; (*Command*)
		Parameter : SystemInputParamter_Type; (*Parameter*)
	END_STRUCT;
	SystemInputCommand_Type : 	STRUCT
		Init : USINT; (*This command initialize all objects of the system*)
		Enable : USINT; (*This command enables all object of the system*)
		Home : USINT; (*This command homes all axes in order defined in the HomeOrder of the axes*)
		ChangeMode : USINT; (*This command changes the mode of the system*)
		EmergencyStop : USINT; (*This command commands a controlled motion stop and transfers the cnc and axes to the state Stopping with the emergency parameters in the cnc and axes daa structure.*)
		Stop : USINT; (*This command commands a controlled motion stop and transfers the cnc and axes to the state Stopping.*)
		Reset : USINT; (*This command makes a transition in the State Diagram from Errorstop to Standstill or Disabled by resetting all internal object errors.*)
		Acknowledge : USINT; (*This command is used to acknowledge the current objects errors.*)
		StartService : USINT; (*This command sets the system into service mode. Global control of the single objects is deactivated*)
		StopService : USINT; (*This command makes a transition in the State Diaram from Service to Disabled or Standstill.*)
		StartSimulation : USINT; (*This command can be used to stwitch the simulation on (SIMULATE_CNC or SIMULATE_MOTOR). *)
		StopSimulation : USINT; (*This command can be used to switch the simulation off.*)
	END_STRUCT;
	SystemInputConfigMode_Type : 	STRUCT
		Label : STRING[LABEL_SIZE]; (*Label is the identifier for external use like the visualization.*)
		Cnc : ARRAY[0..MAX_CNC_MINUS_ONE]OF SystemInputConfigModeCnc_Type; (*Cnc configuration*)
		Axes : ARRAY[0..MAX_AX_MINUS_ONE]OF SystemInputConfigModeAxes_Type; (*Axes configuration*)
	END_STRUCT;
	SystemInputConfigModeAxes_Type : 	STRUCT
		Index : USINT; (*Index of the axis in the Axes_typ.*)
		Type : SystemModeAxesTyp_Type; (*Type of the axis:   CNC_AXES / SPINDLE_0_AXES / SPINDLE_1_AXES / SPINDLE_2_AXES / SPINDLE_3_AXES / JOG_AXES / AUXILIARY_AXES / NO_TYPE.*)
		Behavior : SystemInConfModeAxBehav_Type; (*Behaviour of the axis:  HOME_AUTOPOS_AXES / CYCLIC_POSITION_AXES / STOP_AXES / IGNORE_AXES.*)
		ResetJoltTime : BOOL; (*This is a flag to automatically reset jolt time to zero when exiting jogging mode*)
		Visible : BOOL; (*This bit decides if the axes will be visible in the system monitor.*)
	END_STRUCT;
	SystemInputConfigModeCnc_Type : 	STRUCT
		Index : USINT; (*Index of the cnc in the Cnc_typ.*)
		Behavior : SystemInConfModeCncBehav_Type; (*Behaviour of the cnc: STOP_CNC / IGNORE_CNC.*)
		Visible : BOOL; (*This bit decides if the cnc will be visible in the system monitor.*)
	END_STRUCT;
	SystemInputConfigSystemAxes_Type : 	STRUCT
		Index : USINT; (*Index of the axis in the Axes_typ*)
		HomeOrder : USINT; (*Position in the HomeOrder when calling the System.Input.Command.Home*)
		IsSpindle : BOOL; (*Information Flag for Visualizations*)
		IsEncoder : BOOL;
	END_STRUCT;
	SystemInputConfiguration_Type : 	STRUCT
		Active : BOOL; (*This bit determines if an system is part of the application or not.*)
		Label : STRING[LABEL_SIZE]; (*Label is the identifier for external use like the visualization.*)
		SystemPowerAxesIndex : ARRAY[0..MAX_AX_MINUS_ONE]OF USINT; (*Index of the power supply modules*)
		SystemAxes : ARRAY[0..MAX_AX_MINUS_ONE]OF SystemInputConfigSystemAxes_Type; (*Axes basic configuration, which axis are part of the system*)
		SystemCncIndex : ARRAY[0..MAX_CNC_MINUS_ONE]OF USINT; (*Cnc basic configuration, which cnc system is part of the system*)
		Mode : ARRAY[0..MAX_MODE_MINUS_ONE]OF SystemInputConfigMode_Type; (*Mode configuration*)
	END_STRUCT;
	SystemInputParameterSimMode_Type :
		(
		SIMULATE_CNC, (*This mode switches only the cnc into simulation mode*)
		SIMULATE_MOTOR (*This mode switches the axes into simulation mode*)
		);
	SystemInputParamter_Type : 	STRUCT
		Mode : USINT; (* Mode into the system should be changed *)
		Cooling : SystemInputParamterCooling_Type; (* Cooling parameters *)
		Spindle : SystemInputParamterSpindle_Type; (* Spindle parameters *)
		SimulationMode : SystemInputParameterSimMode_Type; (* Simulation mode (SIMULATE_CNC / SIMULATE_MOTOR) *)
		ConfigOk : BOOL; (* Flag from the configuration, it is set when the system configuration was written *)
		AxesAddress : UDINT; (* Address of the axes structure *)
		CncAddress : UDINT; (* Address of the cnc structure *)
		CommandID : USINT; (* CommandID for axes or cnc commands from the system automaticly increased to be to differ betweeen the different systems *)
	END_STRUCT;
	SystemInputParamterCooling_Type : 	STRUCT
		Mode : SystemInputParamterMode_Type; (* Cooling mode ( FORCE_ON / FORCE_OFF / PROGRAM_DEPENDED ) *)
	END_STRUCT;
	SystemInputParamterMode_Type :
		(
		FORCE_OFF, (* Cooling or spindles are forced off  *)
		FORCE_ON, (* Colling or spindles are forced on *)
		PROGRAM_DEPENDED (* Cooling or spindles are running program depended *)
		);
	SystemInputParamterSpindle_Type : 	STRUCT
		Mode : SystemInputParamterMode_Type; (* Spindle mode ( FORCE_ON / FORCE_OFF / PROGRAM_DEPENDED ) *)
		SpindleVelocity : ARRAY[0..3]OF REAL; (* Spindle velocities for the mode PROGRAM_DEPENDED *)
		Override : REAL; (* Spindle override *)
	END_STRUCT;
	SystemModeAxesTyp_Type :
		(
		NO_TYPE, (* The axes have no type *)
		CNC_AXES, (* The axes with that type get their position from the cnc system ( relative, absolute ... coordinates ) *)
		SPINDLE_0_AXES, (* The axes with that type are spindle0 axes depending movements on the spindle mode and s0 word of the cnc system *)
		SPINDLE_1_AXES, (* The axes with that type are spindle1 axes depending movements on the spindle mode and s1 word of the cnc system *)
		SPINDLE_2_AXES, (* The axes with that type are spindle2 axes depending movements on the spindle mode and s2 word of the cnc system *)
		SPINDLE_3_AXES, (* The axes with that type are spindle3 axes depending movements on the spindle mode and s3 word of the cnc system *)
		JOG_AXES, (* The axes with that type are jogable axes *)
		AUXILIARY_AXES (* The axes with that type are auxiliary axes *)
		);
	SystemOutput_Type : 	STRUCT
		State : SystemOutputState_Type; (* State information *)
		Status : SystemOutputStatus_Type; (* Status information *)
		Monitor : SystemOutputMonitor_Type; (* Monitor information *)
		Error : Error_Type; (* Error information *)
	END_STRUCT;
	SystemOutputMonitor_Type : 	STRUCT
		ModeLabel : STRING[LABEL_SIZE]; (* Actual mode label *)
		Mode : USINT; (* Actual mode index *)
		Cnc : ARRAY[0..MAX_CNC_MINUS_ONE]OF SystemOutputMonitorCnc_Type; (* Cnc monitor information *)
		Axes : ARRAY[0..MAX_AX_MINUS_ONE]OF SystemOutputMonitorAxes_Type; (* Axes monitor information *)
		Cooling : BOOL; (* Cooling status *)
		SpindleMoving : BOOL; (* Spindle status *)
		SpindleMaximalVelocity : REAL; (* Maximal spindle information *)
		SystemAddress : UDINT; (* Address of the system (System_Type) *)
	END_STRUCT;
	SystemOutputMonitorAxes_Type : 	STRUCT
		Label : STRING[LABEL_SIZE]; (* Axes label *)
		Index : USINT; (* Axes index (if no axes is active in that mode then the index is NO_PART_OF_SYSTEM) *)
		AxesDatAddress : UDINT; (* Address of axes ACP10AXIS_typ *)
		Type : SystemModeAxesTyp_Type; (* Axes Type (CNC_AXES / SPINDLE_0_AXES / SPINDLE_1_AXES / SPINDLE_2_AXES / SPINDLE_3_AXES / JOG_AXES / AUXILIARY_AXES / NO_TYPE) *)
		IsSpindle : BOOL; (* Spindle flag for visualization *)
		ActualPostion : REAL; (* Actual position depends of the type *)
		UnitPositionLabel : STRING[LABEL_SIZE]; (* Label of the axis position unit *)
		ActualVelocity : REAL; (* Actual velocity *)
		UnitVelocityLabel : STRING[LABEL_SIZE]; (* Label of the axis velocity unit *)
	END_STRUCT;
	SystemOutputMonitorCnc_Type : 	STRUCT
		Active : BOOL; (* Shows if cnc system is active in the actual mode *)
		Label : STRING[LABEL_SIZE]; (* Label of the cnc system *)
		Index : USINT; (* Index of the cnc system (if no cnc system is active in that mode then the index is NO_PART_OF_SYSTEM) *)
		CncDatAddress : UDINT; (* Address of the cnc system ARNC0CNC_typ *)
	END_STRUCT;
	SystemOutputState_Type : 	STRUCT
		Disabled : BOOL; (* State Disabled see Statediagram *)
		Standby : BOOL; (* State Standby see Statediagram *)
		Homing : BOOL; (* State Homing see Statediagram *)
		Active : BOOL; (* State Active see Statediagram *)
		Stopping : BOOL; (* State Stopping see Statediagram *)
		Errorstop : BOOL; (* State Errorstop see Statediagram *)
		Service : BOOL; (* State Service see Statediagram *)
	END_STRUCT;
	SystemOutputStatus_Type : 	STRUCT
		AccessOk : BOOL; (* All system objects accessed *)
		Busy : BOOL; (* System is busy *)
		HomingOk : BOOL; (* All axes are homed *)
		NetworkInit : BOOL; (* All axes successfulle connected *)
		Booting : BOOL; (* System is booting *)
		Ready : BOOL; (*shows if the controller is ready to be turned on*)
		ControllerStatus : USINT; (*shows if the controllers are all turned on / turned off / not all turned on*)
		CommandError : BOOL; (* System command ignored *)
	END_STRUCT;
END_TYPE
```

### System.var - Local variables
```iecst
(********************************************************************
 * COPYRIGHT -- Bernecker + Rainer
 ********************************************************************
 * Program: System
 * File: System.var
 * Author: radaka
 * Created: February 18, 2009
 ********************************************************************
 * Local variables of program System
 ********************************************************************)
VAR CONSTANT
	CHANGING_MODE : USINT := 253;
	NO_MODE_ACTIVE : USINT := 254;
	NO_PART_OF_SYSTEM : USINT := 254;
	SYSTEM_TIMEOUT : UDINT := 80000;
END_VAR
```

### Program Logical/MotionHandling/SystemHandling/System (IEC) - A new program

#### System.st - Implementation code
```iecst
(********************************************************************
 * COPYRIGHT -- Bernecker + Rainer
 ********************************************************************
 * Program: System
 * File: System.st
 * Author: radaka
 * Created: February 18, 2009
 ********************************************************************
 * Implementation of program System
 ********************************************************************)

PROGRAM _INIT

	StartUpFirst:= 1;

END_PROGRAM

PROGRAM _CYCLIC

	(*************************************************************************************************************)
	(* StartUpFirst routine *)
	IF(StartUpFirst)THEN

		(* Loop over all systems *)
		FOR i:= 0 TO MAX_SYS_MINUS_ONE DO

			pSystem ACCESS ADR(System[i]);

			pSystemPrivate ACCESS ADR(SystemPrivate[i]);

			pSystem.Output.Monitor.SystemAddress:= ADR(System[i]);

		  (* Initialization of Enum Types *)
			pSystemPrivate.TimeoutStep:= SYSTIMEOUTSTEP_CHECK;
			pSystemPrivate.SystemStateStep:= SYSSTATESTEP_BOOTING;
			pSystemPrivate.ActionRequest:= SYSACTION_NO_ACTION;
			pSystemPrivate.ActionResponse:= SYSACTION_NO_ACTION;
			pSystemPrivate.ActionStep:= SYSACTIONSTEP_COMMAND;
			pSystemPrivate.ModeChangeStep:= SYSMODECHANGE_STOP_CNC;
			pSystem.Output.Monitor.Mode:= NO_MODE_ACTIVE;

		(* End Loop over all systems *)
		END_FOR

		StartUpFirst:= 0;
		StartUp:= 1;

	(*************************************************************************************************************)
	(* StartUp routine *)
	ELSIF(StartUp = 1)THEN

		StartUp:= 0;

		(* Loop over all systems *)
		FOR i:= 0 TO MAX_SYS_MINUS_ONE DO

			pSystem ACCESS ADR(System[i]);

			pSystemPrivate ACCESS ADR(SystemPrivate[i]);

			pSystem.Input.Parameter.CommandID:= UDINT_TO_USINT(i + 1);

			pSystem.Input.Parameter.AxesAddress:= System[0].Input.Parameter.AxesAddress;
		 	pSystem.Input.Parameter.CncAddress:= System[0].Input.Parameter.CncAddress;
			pSystem.Input.Parameter.ConfigOk:= System[0].Input.Parameter.ConfigOk;

			IF	(pSystem.Input.Parameter.AxesAddress <> 0)AND
		 		(pSystem.Input.Parameter.CncAddress <> 0)AND
		  		(pSystem.Input.Parameter.ConfigOk = 1)THEN

		 		pAxes ACCESS System[i].Input.Parameter.AxesAddress;
				pCnc ACCESS System[i].Input.Parameter.CncAddress;

			ELSE

				StartUp:= 1;
				RETURN;

		  	END_IF

		(* End loop over all Systems *)
		END_FOR

	ELSE
	(* End StartUp routine *)
	(*************************************************************************************************************)

	(*************************************************************************************************************)
	(* Cyclic routine *)

		(* Loop over all systems *)
		FOR i:= 0 TO MAX_SYS_MINUS_ONE DO

			pSystem ACCESS ADR(System[i]);

			pSystemPrivate ACCESS ADR(SystemPrivate[i]);

			IF(pSystem.Input.Configuration.Active = 1)THEN

				SystemAccess;

				IF(pSystem.Output.Status.AccessOk = 1)THEN

					IF(pSystemPrivate.StartupOk = 0)THEN

						SystemTimeout;

						pSystem.Output.Monitor.Mode:= NO_MODE_ACTIVE;
						pSystem.Output.Monitor.ModeLabel:= 'System booting';
						pSystem.Output.Status.Booting:= 1;

					ELSIF(pSystemPrivate.StartupOk = 1)THEN

						SystemStateHandling;

						SystemActions;

						SystemModechange;

						SystemResetCommands;

						SystemMonitor;

						SystemSpindleHandling;

						SystemCoolingHandling;

						SystemStatus;

					END_IF

				(* End IF(pSystem.Input.Configuration.Active = 1)THEN *)
				END_IF

			(* IF(pSystem.Input.Configuration.Active = 1)THEN *)
			END_IF

		(* End Loop over all systems *)
		END_FOR

	(* End Cyclic routine *)
	(*************************************************************************************************************)
	END_IF

END_PROGRAM
```

#### SystemPrv.typ
```iecst
(********************************************************************
 * COPYRIGHT -- Bernecker + Rainer
 ********************************************************************
 * Program: System
 * File: System.typ
 * Author: radaka
 * Created: February 18, 2009
 ********************************************************************
 * Local data types of program System
 ********************************************************************)

TYPE
	SystemModeChangeSteps_Type :
		(
		SYSMODECHANGE_STOP_CNC,
		SYSMODECHANGE_W_STOP_CNC,
		SYSMODECHANGE_STOP_AXES,
		SYSMODECHANGE_W_STOP_AXES,
		SYSMODECHANGE_HOME_AUTOPOS,
		SYSMODECHANGE_W_HOME_AUTOPOS,
		SYSMODECHANGE_MOVE_AUTOPOS,
		SYSMODECHANGE_W_MOVE_AUTOPOS,
		SYSMODECHANGE_MOVEHOME_AUTOPOS,
		SYSMODECHANGE_W_MOVEHOME_AUTOPOS,
		SYSMODECHANGE_CYCLIC_POSITION,
		SYSMODECHANGE_W_CYCLIC_POSITION,
		SYSMODECHANGE_RESET_JOLT_TIME,
		SYSMODECHANGE_W_RESET_JOLT_TIME,
		SYSMODECHANGE_SET_MODE
		);
	SystemStateSteps_Type :
		(
		SYSSTATESTEP_BOOTING,
		SYSSTATESTEP_DISABLED,
		SYSSTATESTEP_STANDBY,
		SYSSTATESTEP_ACTIVE,
		SYSSTATESTEP_HOMING,
		SYSSTATESTEP_STOPPING,
		SYSSTATESTEP_ERRORSTOP,
		SYSSTATESTEP_SERVICE
		);
	SystemTimeoutSteps_Type :
		(
		SYSTIMEOUTSTEP_CHECK,
		SYSTIMEOUTSTEP_ERROR,
		SYSTIMEOUTSTEP_FINISHED
		);
	SystemActionSteps_Type :
		(
		SYSACTIONSTEP_COMMAND,
		SYSACTIONSTEP_ENABLE_PWR_AXES,
		SYSACTIONSTEP_W_ENABLE_PWR_AXES,
		SYSACTIONSTEP_ENABLE_AXES,
		SYSACTIONSTEP_W_ENABLE_AXES,
		SYSACTIONSTEP_ENABLE_CNC,
		SYSACTIONSTEP_W_ENABLE_CNC,
		SYSACTIONSTEP_ESTOP_CNC,
		SYSACTIONSTEP_W_ESTOP_CNC,
		SYSACTIONSTEP_ESTOP_AXES,
		SYSACTIONSTEP_W_ESTOP_AXES,
		SYSACTIONSTEP_DISABLE_AXES_CNC,
		SYSACTIONSTEP_W_DISABLE_AXES_CNC,
		SYSACTIONSTEP_DISABLE_PWR_AXES,
		SYSACTIONSTEP_HOMING,
		SYSACTIONSTEP_W_HOMING,
		SYSACTIONSTEP_STOPPING_CNC,
		SYSACTIONSTEP_W_STOPPING_CNC,
		SYSACTIONSTEP_STOPPING_AXES,
		SYSACTIONSTEP_W_STOPPING_AXES,
		SYSACTIONSTEP_RESET,
		SYSACTIONSTEP_W_RESET,
		SYSACTIONSTEP_ACKNOWLEDGE,
		SYSACTIONSTEP_INIT,
		SYSACTIONSTEP_W_INIT,
		SYSACTIONSTEP_START_SIMULATION,
		SYSACTIONSTEP_W_START_SIMULATION,
		SYSACTIONSTEP_STOP_SIMULATION,
		SYSACTIONSTEP_W_STOP_SIMULATION
		);
	SystemAction_Type :
		(
		SYSACTION_NO_ACTION,
		SYSACTION_ENABLE,
		SYSACTION_EMERGENCYSTOP,
		SYSACTION_HOME,
		SYSACTION_CHANGEMODE,
		SYSACTION_STOP,
		SYSACTION_RESET,
		SYSACTION_ACKNOWLEDGE,
		SYSACTION_INIT,
		SYSACTION_START_SIMULATION,
		SYSACTION_STOP_SIMULATION
		);
	SystemSpindleHandling_Type : 	STRUCT
		Velocity : REAL;
		ChangeSpeed : BOOL;
		Stop : BOOL;
		Anticlockwise : BOOL;
	END_STRUCT;
	SystemPrivate_Type : 	STRUCT
		SystemStateStep : SystemStateSteps_Type;
		AccessOk : BOOL;
		TimeoutTimer : UDINT;
		TimeoutStep : SystemTimeoutSteps_Type;
		StartupOk : BOOL;
		ActionStep : SystemActionSteps_Type;
		ActionRequest : SystemAction_Type;
		ActionResponse : SystemAction_Type;
		WasEnable : BOOL;
		Disabeling : BOOL;
		Enabeling : BOOL;
		Resetting : BOOL;
		ErrorStopping : BOOL;
		ModeChangeStep : SystemModeChangeSteps_Type;
		ModeChanging : BOOL;
		SpindleHandling : ARRAY[0..3] OF SystemSpindleHandling_Type;
		HomeOrderIndex : USINT;
		HomeFromActive : BOOL;
		OldMode : USINT;
		TempControllerOnStatus : BOOL;
	END_STRUCT;
END_TYPE
```

#### SystemPrv.var
```iecst
(********************************************************************
 * COPYRIGHT -- Bernecker + Rainer
 ********************************************************************
 * Program: System
 * File: SystemPrivate.var
 * Author: radaka
 * Created: February 18, 2009
 ********************************************************************
 * Local variables of program System
 ********************************************************************)
VAR
	System : ARRAY[0..MAX_SYS_MINUS_ONE] OF System_Type := [MAX_SYS_MINUS_ONE+1(0)];
	SystemPrivate : ARRAY[0..MAX_SYS_MINUS_ONE] OF SystemPrivate_Type := [MAX_SYS_MINUS_ONE+1(0)];
	k : UDINT := 0;
	j : UDINT := 0;
	i : UDINT := 0;
	RTInfo_0 : RTInfo := (0);
	pCnc : REFERENCE TO ARRAY[0..MAX_CNC_MINUS_ONE] OF Cnc_Type;
	pAxes : REFERENCE TO ARRAY[0..MAX_AX_MINUS_ONE] OF Axes_Type;
	StartUp : BOOL;
	m : USINT;
	pCncMFunction : REFERENCE TO ARRAY[0..1023] OF USINT;
	n : UDINT;
	TempIndex : USINT;
	TempMode : USINT;
	pSystem : REFERENCE TO System_Type;
	pSystemPrivate : REFERENCE TO SystemPrivate_Type;
	StartUpFirst : BOOL;
	pCncDat : REFERENCE TO ARNC0CNC_typ;
	AxesErrorIndex : STRING[40] := '';
	TempIndexString : STRING[4];
	CncErrorIndex : STRING[40];
	pAxisDat : REFERENCE TO ACP10AXIS_typ;
END_VAR
```
